FUNCTION_BLOCK Q_ChangeObjectLabel (* Command Change Object Label( Part 6 - F.50 ) *)
  (* Standard: ISO 11783-6; Description: This command is used by an ECU to change a label of an object. See also B.21 Object Label Reference List object. Return values iso_s16 - E_NO_ERR - OK - E_OVERFLOW - buffer overflow - E_NOACT - Command not possible in current state - E_NO_INSTANCE - No VT client available *)
  (* Version 1.0, 2022-07-08, franz *)
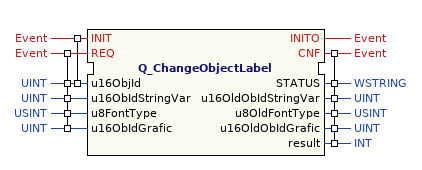
  EVENT_INPUT
    INIT WITH u16ObjId; (* Service Initialization *)
    REQ WITH u16ObjId, u16ObIdStringVar, u8FontType, u16ObIdGrafic; (* Service Request *)
  END_EVENT
  EVENT_OUTPUT
    INITO; (* Initialization Confirm *)
    CNF WITH STATUS, u16OldObIdStringVar, u8OldFontType, u16OldObIdGrafic, result, u16OldObIdStringVar, u8OldFontType, u16OldObIdGrafic; (* Confirmation of Requested Service *)
  END_EVENT
  VAR_INPUT
    u16ObjId : UINT; (* Object ID *)
    u16ObIdStringVar : UINT; (* Object ID of a String Variable object that contains the label string (32 characters maximum) or FFFF if no text is supplied *)
    u8FontType : USINT; (* Font type (ignored if String Variable object reference is NULL or the string contains a WideString ) *)
    u16ObIdGrafic : UINT; (* Object ID of an object to be used as a graphic representation of the object label or FFFF16 if no designator supplied *)
  END_VAR
  VAR_OUTPUT
    STATUS : WSTRING; (* Service Status *)
    u16OldObIdStringVar : UINT; (* Old Object ID of a String Variable object that contains the label string (32 characters maximum) or FFFF if no text is supplied *)
    u8OldFontType : USINT; (* Old value for attribute *)
    u16OldObIdGrafic : UINT;
    result : INT; (* retval see description *)
  END_VAR
END_FUNCTION_BLOCK
